// TwinCAT 3 PLC project PLC_MASTER
// ProgramVersion: 3.1.4026.16
// libraries:
//   Tc2_Standard, * (Beckhoff Automation GmbH)
//   Tc2_System, * (Beckhoff Automation GmbH)
// project tree:
//   / PlcTask.TcTTO
//   POUs/ MAIN.TcPOU
// real-time tasks:
//   TASK PlcTask: cycle T#10ms, priority 20, ADS port 350
// I/O:
//   DEVICE Device 1 (EtherCAT), AmsNetId 10.200.70.9.2.1
//     Box 1 (CX5140 EtherCAT slave) [CX5140 EtherCAT slave]
//     Box 2 (CX5140 EtherCAT slave) [CX5140 EtherCAT slave]
// variable links:
//   PLC_MASTER Instance <-> Device 1 (EtherCAT)/Box 1 (CX5140 EtherCAT slave)
//     PlcTask Inputs/MAIN.bFlag1 <-> IO Inputs/bFlag
//     PlcTask Inputs/MAIN.iSlaveCounter1 <-> IO Inputs/iSlaveCounter
//     PlcTask Inputs/MAIN.lrSlaveTemp1 <-> IO Inputs/lrSlaveTemp
//     PlcTask Outputs/MAIN.bTrigger <-> IO Outputs/bTrigger
//     PlcTask Outputs/MAIN.iMasterCounter <-> IO Outputs/iMasterCounter
//     PlcTask Outputs/MAIN.lrMasterTemp <-> IO Outputs/lrMasterTemp
//   PLC_MASTER Instance <-> Device 1 (EtherCAT)/Box 2 (CX5140 EtherCAT slave)
//     PlcTask Inputs/MAIN.bFlag2 <-> IO Inputs/bFlag
//     PlcTask Inputs/MAIN.iSlaveCounter2 <-> IO Inputs/iSlaveCounter
//     PlcTask Inputs/MAIN.lrSlaveTemp2 <-> IO Inputs/lrSlaveTemp
//     PlcTask Outputs/MAIN.bTrigger <-> IO Outputs/bTrigger
//     PlcTask Outputs/MAIN.iMasterCounter <-> IO Outputs/iMasterCounter
//     PlcTask Outputs/MAIN.lrMasterTemp <-> IO Outputs/lrMasterTemp

CONFIGURATION PLC_MASTER
    RESOURCE PLC ON TwinCAT3
        TASK PlcTask(INTERVAL := T#10ms, PRIORITY := 20);
        PROGRAM MAIN WITH PlcTask : MAIN;
    END_RESOURCE
END_CONFIGURATION

// ---- POUs/MAIN.TcPOU
PROGRAM MAIN//EtherCAT Master side
VAR
	iMasterCounter 	AT %Q* : INT;	//integer 	input from Master
	lrMasterTemp 	AT %Q* : LREAL;	//lreal		input from Master
	bTrigger 		AT %Q* : BOOL;	//bool 		input from Master
	
	iSlaveCounter1 	AT %I* : INT;	//integer	output to Master
	lrSlaveTemp1 	AT %I* : LREAL;	//lreal		output to Master
	bFlag1 			AT %I* : BOOL;	//bool		output to Master
	iSlaveCounter2 	AT %I* : INT;	//integer	output to Master
	lrSlaveTemp2 	AT %I* : LREAL;	//lreal		output to Master
	bFlag2 			AT %I* : BOOL;	//bool		output to Master

	lag1,lag2: INT;
END_VAR

//EtherCAT Master side
lag1:=iMasterCounter-iSlaveCounter1;
lag2:=iMasterCounter-iSlaveCounter2;

iMasterCounter:= iMasterCounter+1;
lrMasterTemp;
bTrigger;

iSlaveCounter1;
lrSlaveTemp1;
bFlag1;

iSlaveCounter2;
lrSlaveTemp2;
bFlag2;

END_PROGRAM
